PROGRAM MAIN
VAR
END_VAR

END_PROGRAM

(* stored: Version 1.1.0.1
   POU MAIN: Id {8f5954ce-d17e-4752-94a4-9ae2de0eb458} *)
